// Mitsubishi GX Works2 project: luukhoremakev4   PLC: FX1N/FX1NC
// mainchinh

PROGRAM MAIN
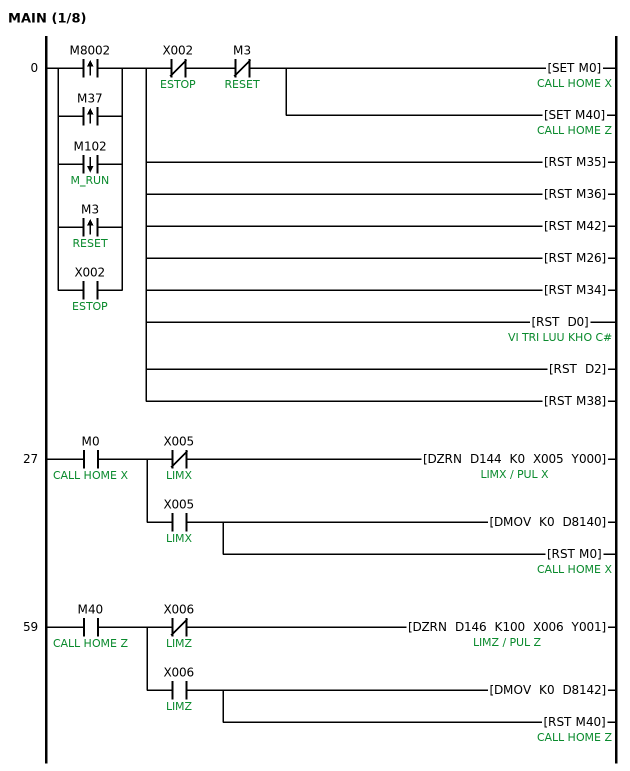
0     LDP     M8002
      ORP     M37
      ORF     M102  ; M_RUN
      ORP     M3  ; RESET
      OR      X002  ; ESTOP
      MPS
      ANI     X002  ; ESTOP
      ANI     M3  ; RESET
      SET     M0  ; CALL HOME X
      SET     M40  ; CALL HOME Z
      MPP
      RST     M35
      RST     M36
      RST     M42
      RST     M26
      RST     M34
      RST     D0  ; VI TRI LUU KHO C#
      RST     D2
      RST     M38
27    LD      M0  ; CALL HOME X
      MPS
      ANI     X005  ; LIMX
      DZRN    D144 K0 X005 Y000  ; PUL X
      MPP
      AND     X005  ; LIMX
      DMOV    K0 D8140
      RST     M0  ; CALL HOME X
59    LD      M40  ; CALL HOME Z
      MPS
      ANI     X006  ; LIMZ
      DZRN    D146 K100 X006 Y001  ; PUL Z
      MPP
      AND     X006  ; LIMZ
      DMOV    K0 D8142
      RST     M40  ; CALL HOME Z
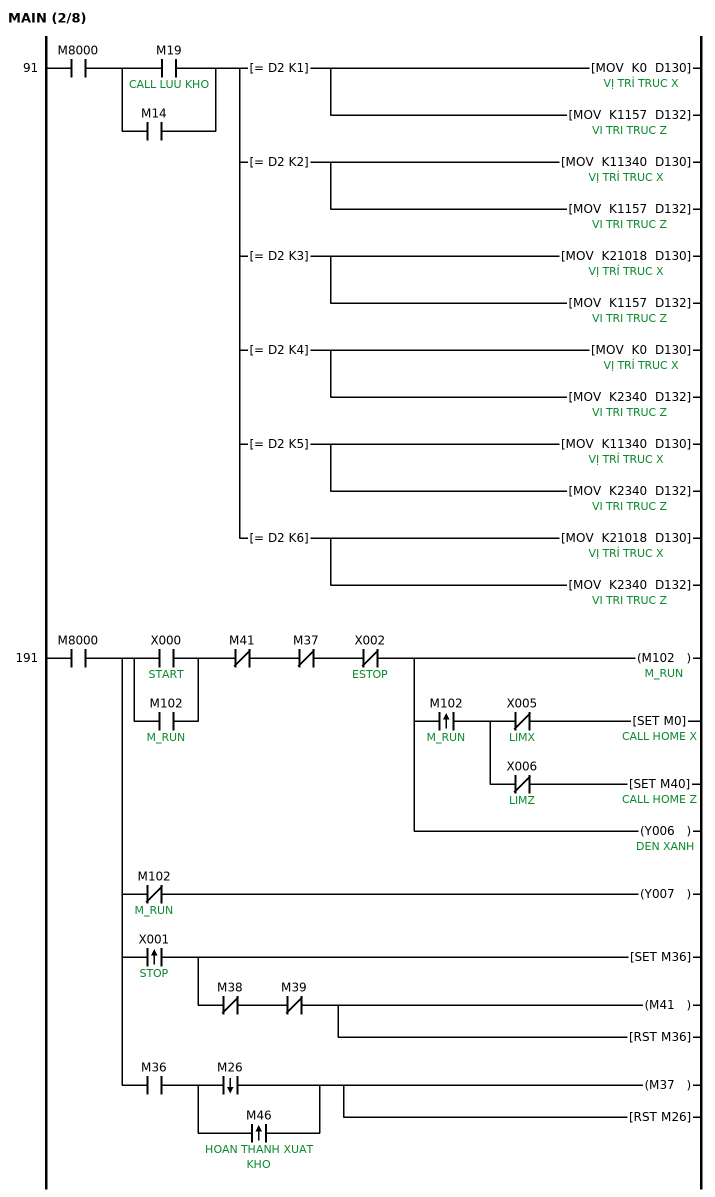
91    LD      M8000
      LD      M19  ; CALL LUU KHO
      OR      M14
      ANB
      MPS
      AND=    D2 K1
      MOV     K0 D130  ; VỊ TRÍ TRUC X
      MOV     K1157 D132  ; VI TRI TRUC Z
      MRD
      AND=    D2 K2
      MOV     K11340 D130
      MOV     K1157 D132
      MRD
      AND=    D2 K3
      MOV     K21018 D130
      MOV     K1157 D132
      MRD
      AND=    D2 K4
      MOV     K0 D130
      MOV     K2340 D132
      MRD
      AND=    D2 K5
      MOV     K11340 D130
      MOV     K2340 D132
      MPP
      AND=    D2 K6
      MOV     K21018 D130
      MOV     K2340 D132
191   LD      M8000
      MPS
      LD      X000  ; START
      OR      M102  ; M_RUN
      ANB
      ANI     M41
      ANI     M37
      ANI     X002  ; ESTOP
      OUT     M102  ; M_RUN
      MPS
      ANDP    M102  ; M_RUN
      MPS
      ANI     X005  ; LIMX
      SET     M0  ; CALL HOME X
      MPP
      ANI     X006  ; LIMZ
      SET     M40  ; CALL HOME Z
      MPP
      OUT     Y006  ; DEN XANH
      MRD
      ANI     M102  ; M_RUN
      OUT     Y007
      MRD
      ANDP    X001  ; STOP
      SET     M36
      ANI     M38
      ANI     M39
      OUT     M41
      RST     M36
      MPP
      AND     M36
      LDF     M26
      ORP     M46  ; HOAN THANH XUAT KHO
      ANB
      OUT     M37
      RST     M26
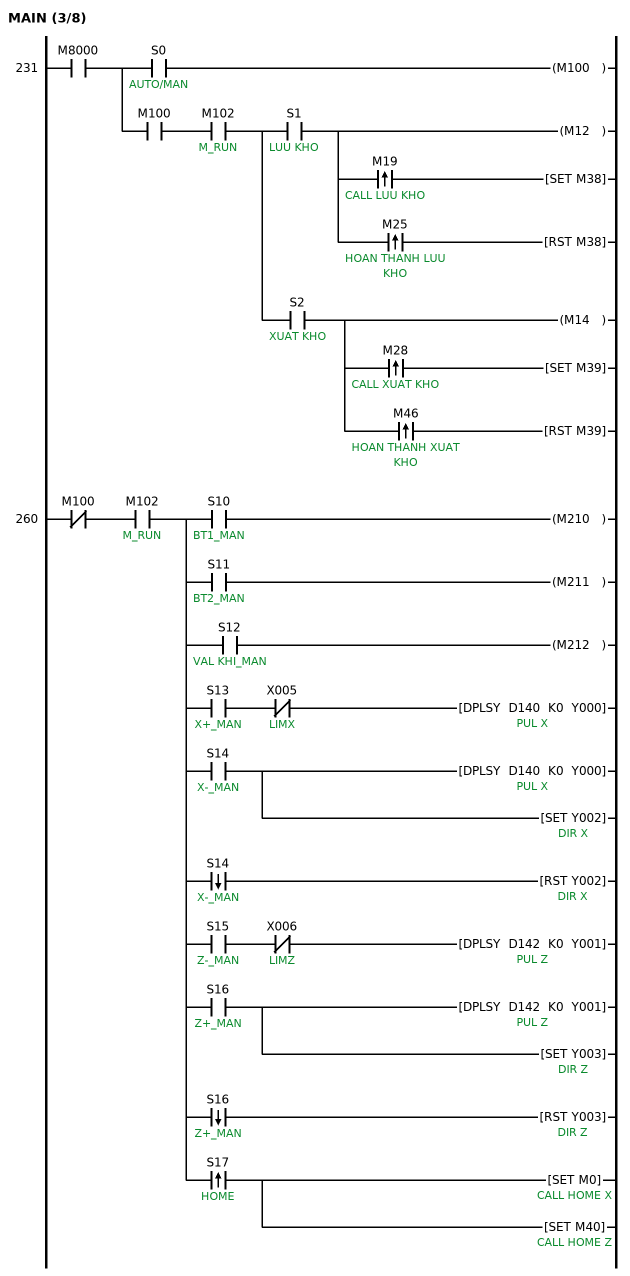
231   LD      M8000
      MPS
      AND     S0  ; AUTO/MAN
      OUT     M100
      MPP
      AND     M100
      AND     M102  ; M_RUN
      MPS
      AND     S1  ; LUU KHO
      OUT     M12
      MPS
      ANDP    M19  ; CALL LUU KHO
      SET     M38
      MPP
      ANDP    M25  ; HOAN THANH LUU KHO
      RST     M38
      MPP
      AND     S2  ; XUAT KHO
      OUT     M14
      MPS
      ANDP    M28  ; CALL XUAT KHO
      SET     M39
      MPP
      ANDP    M46  ; HOAN THANH XUAT KHO
      RST     M39
260   LDI     M100
      AND     M102  ; M_RUN
      MPS
      AND     S10  ; BT1_MAN
      OUT     M210
      MRD
      AND     S11  ; BT2_MAN
      OUT     M211
      MRD
      AND     S12  ; VAL KHI_MAN
      OUT     M212
      MRD
      AND     S13  ; X+_MAN
      ANI     X005  ; LIMX
      DPLSY   D140 K0 Y000
      MRD
      AND     S14  ; X-_MAN
      DPLSY   D140 K0 Y000
      SET     Y002  ; DIR X
      MRD
      ANDF    S14  ; X-_MAN
      RST     Y002  ; DIR X
      MRD
      AND     S15  ; Z-_MAN
      ANI     X006  ; LIMZ
      DPLSY   D142 K0 Y001
      MRD
      AND     S16  ; Z+_MAN
      DPLSY   D142 K0 Y001
      SET     Y003  ; DIR Z
      MRD
      ANDF    S16  ; Z+_MAN
      RST     Y003  ; DIR Z
      MPP
      ANDP    S17  ; HOME
      SET     M0  ; CALL HOME X
      SET     M40  ; CALL HOME Z
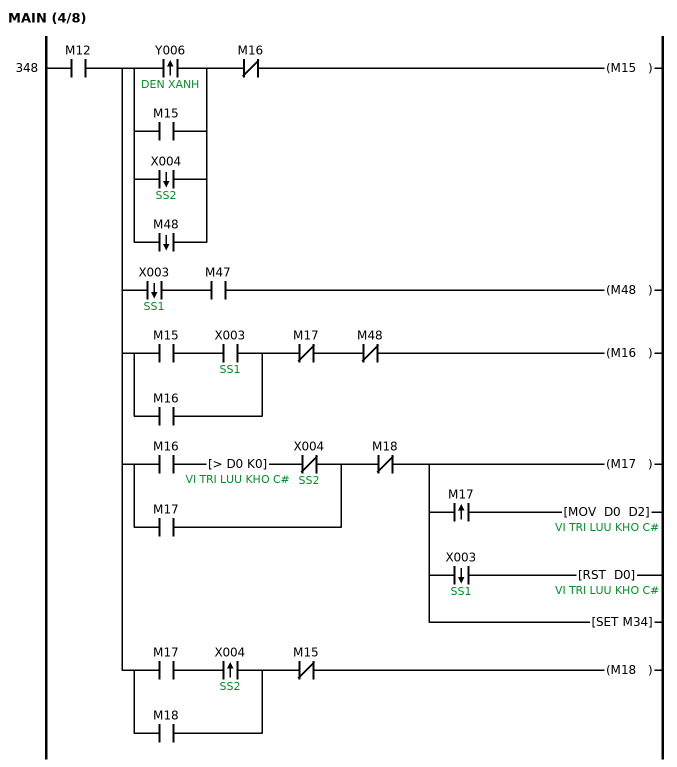
348   LD      M12
      MPS
      LDP     Y006  ; DEN XANH
      OR      M15
      ORF     X004  ; SS2
      ORF     M48
      ANB
      ANI     M16
      OUT     M15
      MRD
      ANDF    X003  ; SS1
      AND     M47
      OUT     M48
      MRD
      LD      M15
      AND     X003  ; SS1
      OR      M16
      ANB
      ANI     M17
      ANI     M48
      OUT     M16
      MRD
      LD      M16
      AND>    D0 K0  ; VI TRI LUU KHO C#
      ANI     X004  ; SS2
      OR      M17
      ANB
      ANI     M18
      OUT     M17
      MPS
      ANDP    M17
      MOV     D0 D2
      MRD
      ANDF    X003  ; SS1
      RST     D0  ; VI TRI LUU KHO C#
      MPP
      SET     M34
      MPP
      LD      M17
      ANDP    X004  ; SS2
      OR      M18
      ANB
      ANI     M15
      OUT     M18
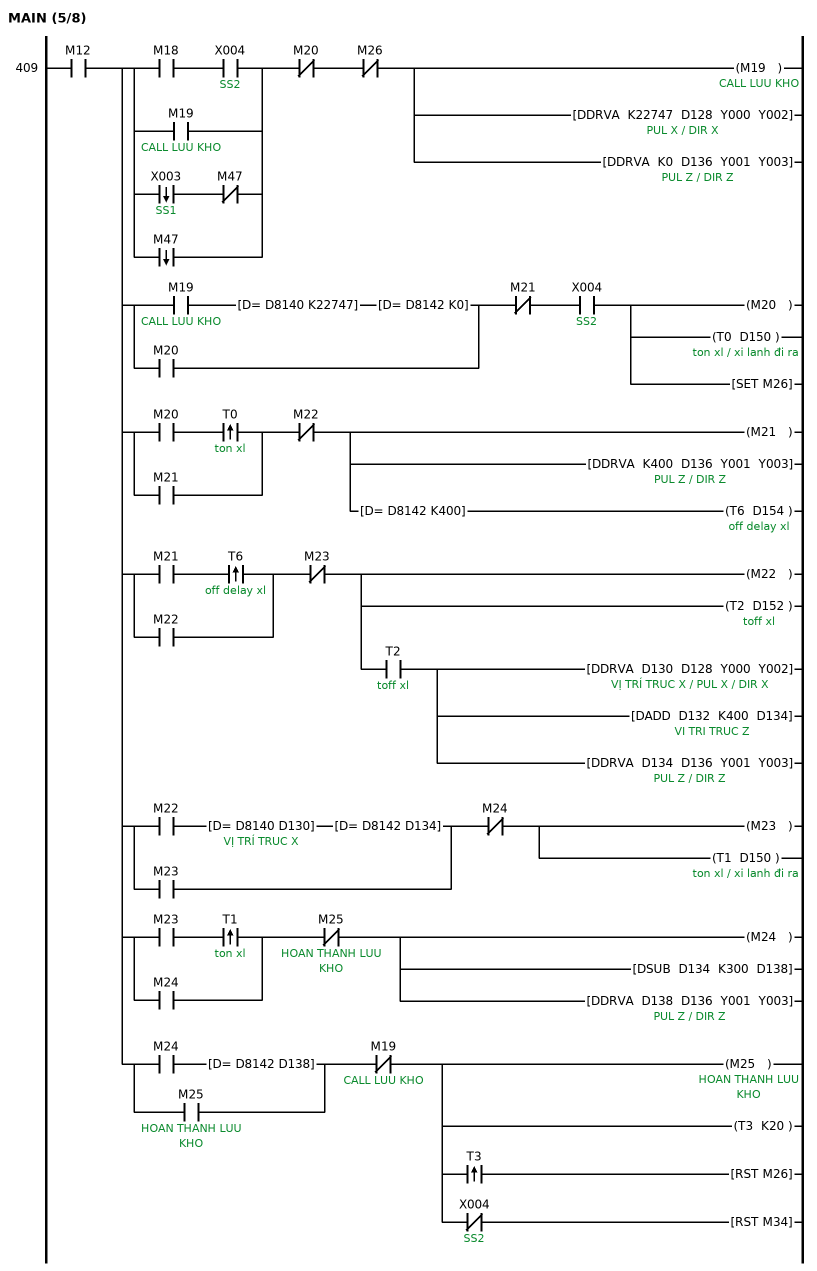
409   LD      M12
      MPS
      LD      M18
      AND     X004  ; SS2
      OR      M19  ; CALL LUU KHO
      LDF     X003  ; SS1
      ANI     M47
      ORB
      ORF     M47
      ANB
      ANI     M20
      ANI     M26
      OUT     M19  ; CALL LUU KHO
        [note] DI CHUYEN DEN VI TRI NHAP/LK
      DDRVA   K22747 D128 Y000 Y002
      DDRVA   K0 D136 Y001 Y003
      MRD
      LD      M19  ; CALL LUU KHO
      ANDD=   D8140 K22747
      ANDD=   D8142 K0
      OR      M20
      ANB
      ANI     M21
      AND     X004  ; SS2
      OUT     M20
      OUT     T0 D150  ; ton xl / xi lanh đi ra
      SET     M26
      MRD
      LD      M20
      ANDP    T0  ; ton xl
      OR      M21
      ANB
      ANI     M22
      OUT     M21
        [note] NANG Z LAY HANG/LK
      DDRVA   K400 D136 Y001 Y003
      ANDD=   D8142 K400
      OUT     T6 D154  ; off delay xl
      MRD
      LD      M21
      ANDP    T6  ; off delay xl
      OR      M22
      ANB
      ANI     M23
      OUT     M22
        [note] DEN VI TRI CAC O HANG/LK
      OUT     T2 D152  ; toff xl
      AND     T2  ; toff xl
      DDRVA   D130 D128 Y000 Y002
      DADD    D132 K400 D134
      DDRVA   D134 D136 Y001 Y003
      MRD
      LD      M22
      ANDD=   D8140 D130  ; VỊ TRÍ TRUC X
      ANDD=   D8142 D134
      OR      M23
      ANB
      ANI     M24
      OUT     M23
      OUT     T1 D150  ; ton xl / xi lanh đi ra
      MRD
      LD      M23
      ANDP    T1  ; ton xl
      OR      M24
      ANB
      ANI     M25  ; HOAN THANH LUU KHO
      OUT     M24
        [note] HA TRUC Z/LK
      DSUB    D134 K300 D138
      DDRVA   D138 D136 Y001 Y003
      MPP
      LD      M24
      ANDD=   D8142 D138
      OR      M25  ; HOAN THANH LUU KHO
      ANB
      ANI     M19  ; CALL LUU KHO
      OUT     M25  ; HOAN THANH LUU KHO
      OUT     T3 K20
      MPS
      ANDP    T3
      RST     M26
      MPP
      ANI     X004  ; SS2
      RST     M34
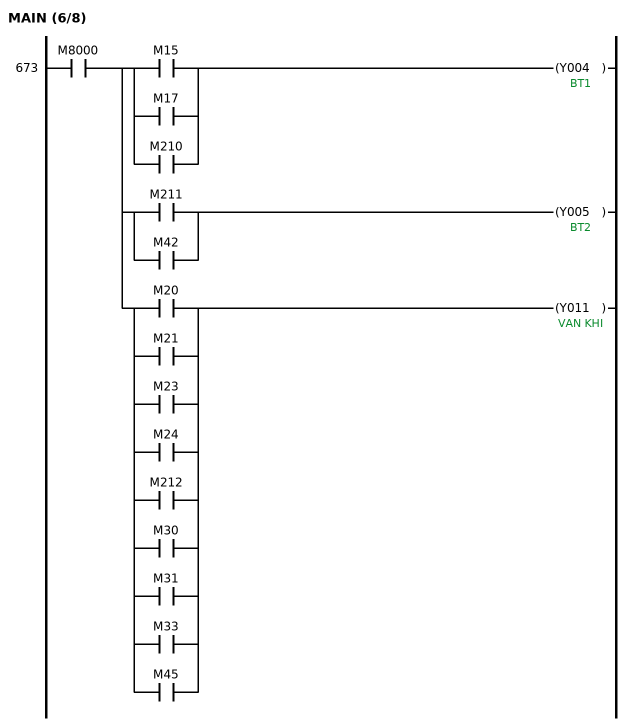
673   LD      M8000
      MPS
      LD      M15
      OR      M17
      OR      M210
      ANB
      OUT     Y004  ; BT1
      MRD
      LD      M211
      OR      M42
      ANB
      OUT     Y005  ; BT2
      MPP
      LD      M20
      OR      M21
      OR      M23
      OR      M24
      OR      M212
      OR      M30
      OR      M31
      OR      M33
      OR      M45
      ANB
      OUT     Y011  ; VAN KHI
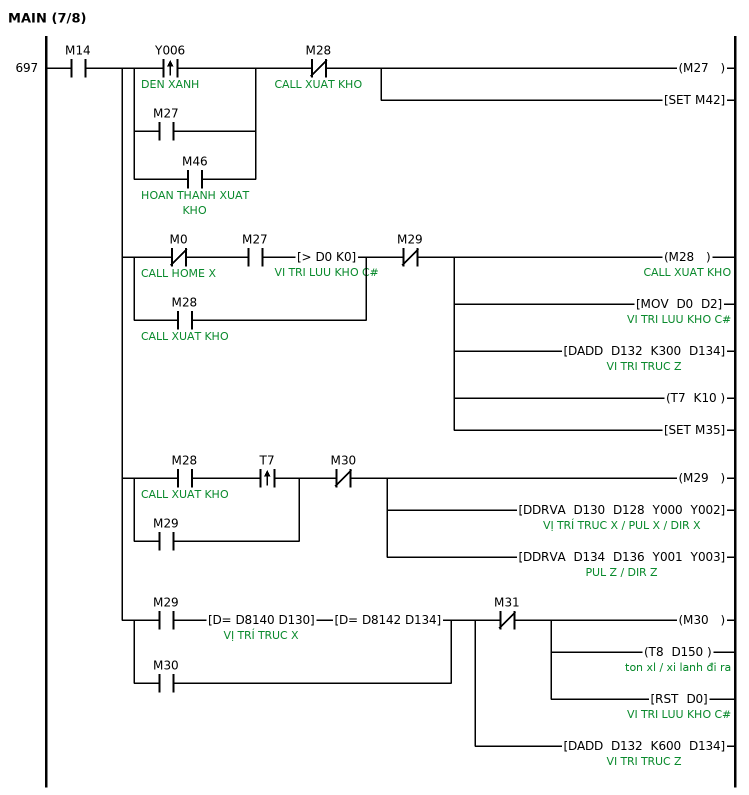
697   LD      M14
      MPS
      LDP     Y006  ; DEN XANH
      OR      M27
      OR      M46  ; HOAN THANH XUAT KHO
      ANB
      ANI     M28  ; CALL XUAT KHO
      OUT     M27
      SET     M42
      MRD
      LDI     M0  ; CALL HOME X
      AND     M27
      AND>    D0 K0  ; VI TRI LUU KHO C#
      OR      M28  ; CALL XUAT KHO
      ANB
      ANI     M29
      OUT     M28  ; CALL XUAT KHO
      MOV     D0 D2
      DADD    D132 K300 D134
        [note] + TRUC Z (O HANG)
      OUT     T7 K10
      SET     M35
      MRD
      LD      M28  ; CALL XUAT KHO
      ANDP    T7
      OR      M29
      ANB
      ANI     M30
      OUT     M29
        [note] DEN VI TRI XUAT/XK
      DDRVA   D130 D128 Y000 Y002
      DDRVA   D134 D136 Y001 Y003
      MPP
      LD      M29
      ANDD=   D8140 D130  ; VỊ TRÍ TRUC X
      ANDD=   D8142 D134
      OR      M30
      ANB
      MPS
      ANI     M31
      OUT     M30
      OUT     T8 D150  ; ton xl / xi lanh đi ra
      RST     D0  ; VI TRI LUU KHO C#
      MPP
      DADD    D132 K600 D134
        [note] +TRUC Z(O HANG)
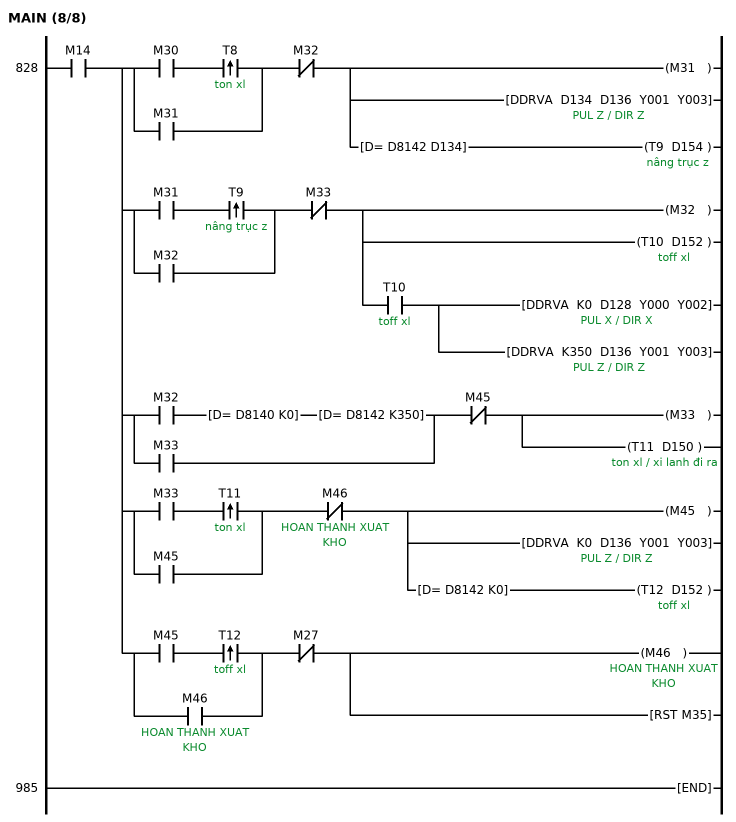
828   LD      M14
      MPS
      LD      M30
      ANDP    T8  ; ton xl
      OR      M31
      ANB
      ANI     M32
      OUT     M31
      DDRVA   D134 D136 Y001 Y003
      ANDD=   D8142 D134
      OUT     T9 D154  ; nâng trục z
      MRD
      LD      M31
      ANDP    T9  ; nâng trục z
      OR      M32
      ANB
      ANI     M33
      OUT     M32
        [note] DEN VI TRI XUAT/XK
      OUT     T10 D152  ; toff xl
      AND     T10  ; toff xl
      DDRVA   K0 D128 Y000 Y002
      DDRVA   K350 D136 Y001 Y003
      MRD
      LD      M32
      ANDD=   D8140 K0
      ANDD=   D8142 K350
      OR      M33
      ANB
      ANI     M45
      OUT     M33
      OUT     T11 D150  ; ton xl / xi lanh đi ra
      MRD
      LD      M33
      ANDP    T11  ; ton xl
      OR      M45
      ANB
      ANI     M46  ; HOAN THANH XUAT KHO
      OUT     M45
        [note] HA TRUC Z/XK
      DDRVA   K0 D136 Y001 Y003
      ANDD=   D8142 K0
      OUT     T12 D152  ; toff xl
      MPP
      LD      M45
      ANDP    T12  ; toff xl
      OR      M46  ; HOAN THANH XUAT KHO
      ANB
      ANI     M27
      OUT     M46  ; HOAN THANH XUAT KHO
      RST     M35
985   END
END_PROGRAM
